// TIA Portal V20 export
VAR_GLOBAL   // PLC tag table "默认变量表"
   右顶升V90_Drive_IN AT %I68.0 : "PD_TEL3_IN";
   右顶升V90_Drive_OUT AT %Q68.0 : "PD_TEL3_OUT";
   左顶升IS620F_Drive_IN AT %I86.0 : "PD_TEL3_IN";
   左顶升IS620F_Drive_OUT AT %Q78.0 : "PD_TEL3_OUT";
   System_Byte AT %MB1 : Byte;
   FirstScan AT %M1.0 : Bool;
   DiagStatusUpdate AT %M1.1 : Bool;
   AlwaysTRUE AT %M1.2 : Bool;
   AlwaysFALSE AT %M1.3 : Bool;
   Clock_Byte AT %MB0 : Byte;
   Clock_10Hz AT %M0.0 : Bool;
   Clock_5Hz AT %M0.1 : Bool;
   "Clock_2.5Hz" AT %M0.2 : Bool;
   Clock_2Hz AT %M0.3 : Bool;
   "Clock_1.25Hz" AT %M0.4 : Bool;
   Clock_1Hz AT %M0.5 : Bool;
   "Clock_0.625Hz" AT %M0.6 : Bool;
   "Clock_0.5Hz" AT %M0.7 : Bool;
   右顶升V90控制字 AT %MW2 : Word;
   左顶升IS620F控制字 AT %MW4 : Word;
   左_回原模式 AT %MW6 : Int;
   左_绝对位置 AT %MD8 : Real;
   左_绝对速度 AT %MD12 : Real;
   左_相对位置 AT %MD16 : Real;
   左_相对速度 AT %MD20 : Real;
   左_点动速度 AT %MD24 : Real;
   左顶升IS620F状态字 AT %MW28 : Word;
   左顶升当前位置 AT %MD30 : Real;
   左顶升当前速度 AT %MD34 : Real;
   右顶升V90状态字 AT %MW38 : Word;
   右_回原模式 AT %MW40 : Int;
   右_绝对位置 AT %MD42 : Real;
   右_绝对速度 AT %MD46 : Real;
   右_相对位置 AT %MD50 : Real;
   右_相对速度 AT %MD54 : Real;
   右_点动速度 AT %MD58 : Real;
   右顶升当前位置 AT %MD62 : Real;
   右顶升当前速度 AT %MD66 : Real;
END_VAR
